FUNCTION alg_a_vacuum : BOOL
VAR_INPUT
	state: STATE;
END_VAR

alg_a_vacuum := FALSE;

END_FUNCTION

(* stored: Version 1.1.0.1, ProductVersion 3.1.4022.18
   POU alg_a_vacuum: Id {6d688531-21f4-434b-afa6-748f464113e2}, SpecialFunc None *)
